FUNCTION_BLOCK FB_Convert_10V2co2
VAR_INPUT
	iInput			:	INT;
	tRefresh		:	TIME;
END_VAR
VAR_OUTPUT
	wOut			:	WORD;
END_VAR
VAR
	rX				:	REAL;
	tonBlock		:	TON;
	bBlock			:	BOOL := FALSE;
END_VAR

// For Convertion of 0-10V Signal from 0-2000ppm
tonBlock(IN := bBlock, PT := tRefresh);

IF NOT bBLock THEN

	rX := iInput * 0.061037018951994; //Annahme 10V entspr. 32767
	wOut := REAL_TO_WORD(rX);

	bBlock := TRUE;
	
END_IF

IF tonBlock.Q THEN
	bBlock := FALSE;
END_IF

END_FUNCTION_BLOCK

(* stored: Version 1.1.0.1, ProductVersion 3.1.4024.4
   POU FB_Convert_10V2co2: Id {2a0fff5a-8a96-4a48-8796-375c2e83e973}, SpecialFunc None *)
